(* Logix 5000 project; controller Oven_and_Boiler_V35 vendor 1 type 14 code 214 rev 38.11; software revision 38.01; part 2 of 2 *)
(* tags used below, declared in another part *)
   ActualSetpoint : DINT;   // Actual temperature setpoint (for current phase)
   ActualTemperature : REAL;
   Gas : REAL;
   GasThrottle : REAL;
   kW : REAL;
   kWh : REAL;
   Preheating : BOOL;
   Running : BOOL;   // Status: Sequence is Running
   SET_PreheatingTemperature : DINT;   // Setpoint: Preheating Temperature
   TotEE : REAL;
   TotLPG : REAL;
   WRK_Gas_change : REAL;
   WRK_kWh_change : REAL;
   WRK_TemperatureSetpoint : REAL;
   WRK_throttle : REAL;
   zCTRL_Timer : TIMER;
   Tank1 : TankUDT;
   Tank1_Level : REAL;
   Tank1_SetPoint : REAL;
   Tank1_ValveInCmd : BOOL;
   Tank1_ValveInStatus : BOOL;
   Tank1_ValveOutCmd : BOOL;
   Tank1_ValveOutStatus : BOOL;
   Tank2 : TankUDT;
   Tank2_Level : REAL;
   Tank2_SetPoint : REAL;
   Tank2_ValveInCmd : BOOL;
   Tank2_ValveInStatus : BOOL;
   Tank2_ValveOutCmd : BOOL;
   Tank2_ValveOutStatus : BOOL;
   Tank3_Level : REAL;
   Tank3_SetPoint : REAL;
   Tank3_ValveInCmd : BOOL;
   Tank3_ValveInStatus : BOOL;
   Tank3_ValveOutCmd : BOOL;
   Tank3_ValveOutStatus : BOOL;
(* OvenDemo, continued *)

ROUTINE OvenTemperature   (* ladder *)
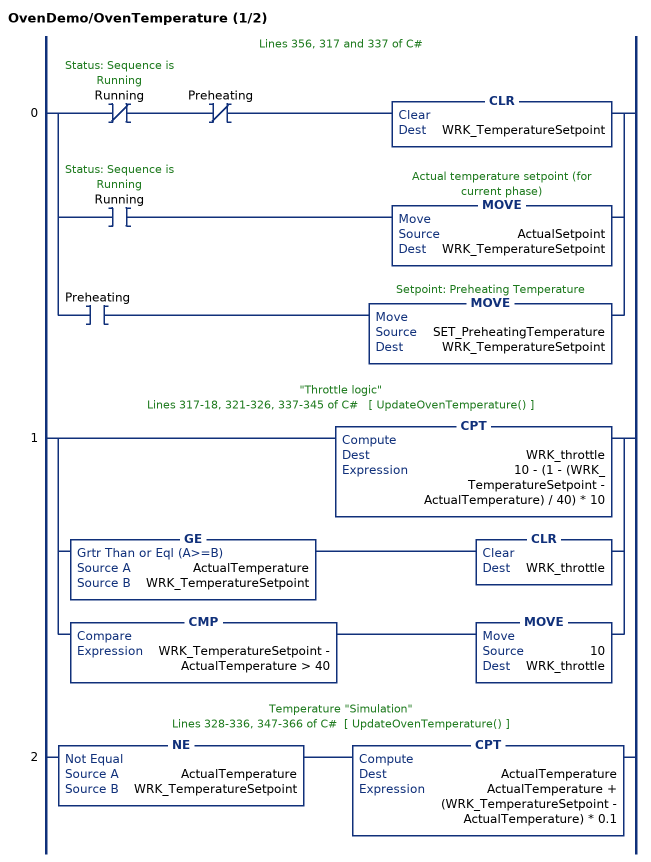
   // Lines 356, 317 and 337 of C#
   0: [XIO(Running) XIO(Preheating) CLR(WRK_TemperatureSetpoint) ,XIC(Running) MOVE(ActualSetpoint,WRK_TemperatureSetpoint) ,XIC(Preheating) MOVE(SET_PreheatingTemperature,WRK_TemperatureSetpoint) ];
   // "Throttle logic"
   // Lines 317-18, 321-326, 337-345 of C#   [ UpdateOvenTemperature() ]
   1: [CPT(WRK_throttle,10 - (1 - (WRK_TemperatureSetpoint - ActualTemperature) / 40) * 10) ,GE(ActualTemperature,WRK_TemperatureSetpoint) CLR(WRK_throttle) ,CMP(WRK_TemperatureSetpoint - ActualTemperature > 40) MOVE(10,WRK_throttle) ];
   // Temperature "Simulation"
   // Lines 328-336, 347-366 of C#  [ UpdateOvenTemperature() ]
   2: NE(ActualTemperature,WRK_TemperatureSetpoint)CPT(ActualTemperature,ActualTemperature + (WRK_TemperatureSetpoint - ActualTemperature) * 0.1);
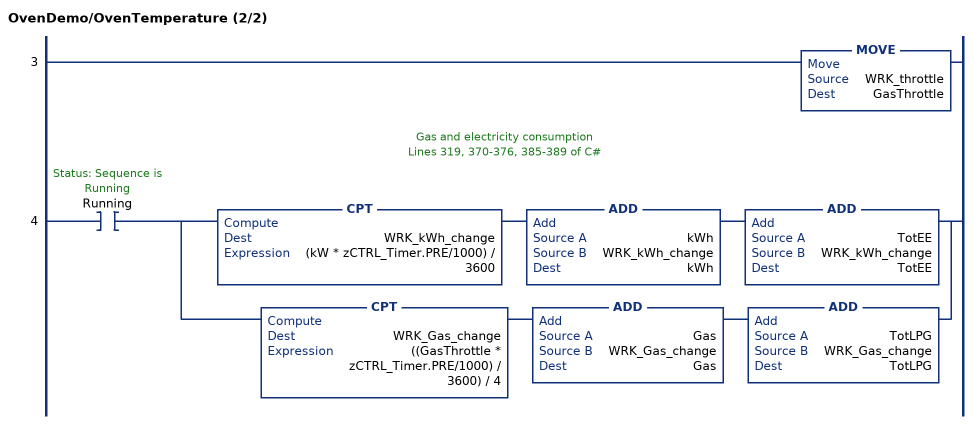
   3: MOVE(WRK_throttle,GasThrottle);
   // Gas and electricity consumption
   // Lines 319, 370-376, 385-389 of C#
   4: XIC(Running)[CPT(WRK_kWh_change,(kW * zCTRL_Timer.PRE/1000) / 3600) ADD(kWh,WRK_kWh_change,kWh) ADD(TotEE,WRK_kWh_change,TotEE) ,CPT(WRK_Gas_change,((GasThrottle * zCTRL_Timer.PRE/1000) / 3600) / 4) ADD(Gas,WRK_Gas_change,Gas) ADD(TotLPG,WRK_Gas_change,TotLPG) ];
END_ROUTINE
END_PROGRAM

PROGRAM TankLogic   (* main routine MainRoutine *)

ROUTINE MainRoutine   (* ladder *)
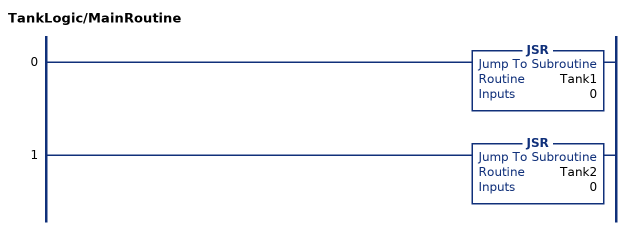
   0: JSR(Tank1,0);
   1: JSR(Tank2,0);
END_ROUTINE

ROUTINE Tank1   (* ladder *)
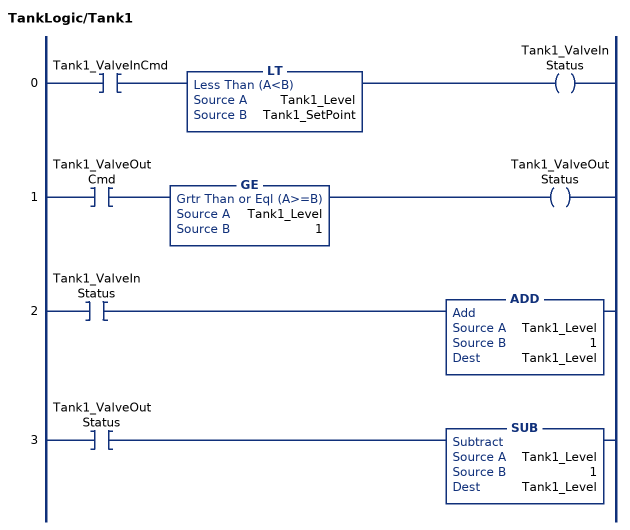
   0: XIC(Tank1_ValveInCmd)LT(Tank1_Level,Tank1_SetPoint)OTE(Tank1_ValveInStatus);
   1: XIC(Tank1_ValveOutCmd)GE(Tank1_Level,1)OTE(Tank1_ValveOutStatus);
   2: XIC(Tank1_ValveInStatus)ADD(Tank1_Level,1,Tank1_Level);
   3: XIC(Tank1_ValveOutStatus)SUB(Tank1_Level,1,Tank1_Level);
END_ROUTINE

ROUTINE Tank2   (* ladder *)
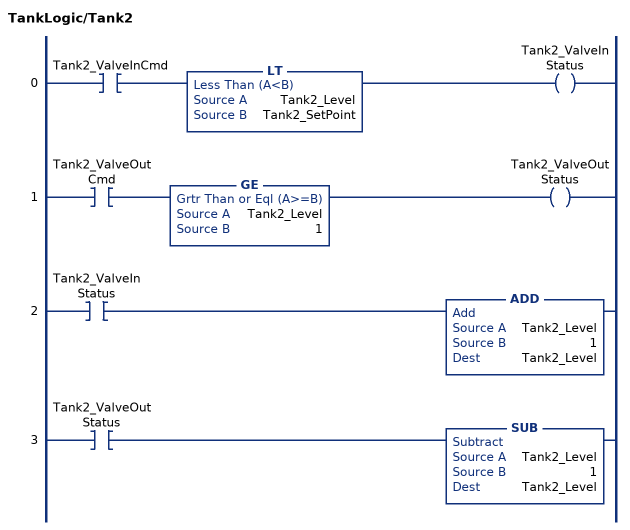
   0: XIC(Tank2_ValveInCmd)LT(Tank2_Level,Tank2_SetPoint)OTE(Tank2_ValveInStatus);
   1: XIC(Tank2_ValveOutCmd)GE(Tank2_Level,1)OTE(Tank2_ValveOutStatus);
   2: XIC(Tank2_ValveInStatus)ADD(Tank2_Level,1,Tank2_Level);
   3: XIC(Tank2_ValveOutStatus)SUB(Tank2_Level,1,Tank2_Level);
END_ROUTINE

ROUTINE Tank3   (* ladder *)
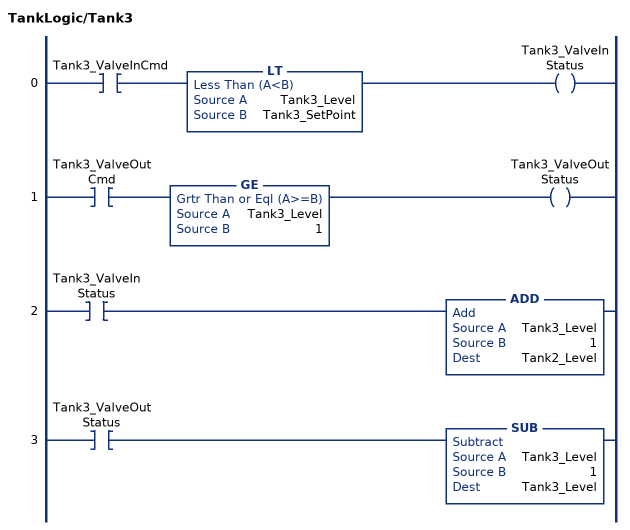
   0: XIC(Tank3_ValveInCmd)LT(Tank3_Level,Tank3_SetPoint)OTE(Tank3_ValveInStatus);
   1: XIC(Tank3_ValveOutCmd)GE(Tank3_Level,1)OTE(Tank3_ValveOutStatus);
   2: XIC(Tank3_ValveInStatus)ADD(Tank3_Level,1,Tank2_Level);
   3: XIC(Tank3_ValveOutStatus)SUB(Tank3_Level,1,Tank3_Level);
END_ROUTINE
END_PROGRAM
